FUNCTION_BLOCK PUBLIC FB_Step EXTENDS FB_Base
VAR_INPUT
END_VAR
VAR_OUTPUT
	nActStep	: UDINT := 0 ; // Active step
	bIdle		: BOOL	:= TRUE  ; // Stepper is idle (Step 0)
	bPaused		: BOOL 	:= FALSE ; // Stepper is paused
	bHold		: BOOL 	:= FALSE ; // Stepper is blocked for changes
	bSkipPause	: BOOL	:= FALSE ; // Pause function is skipped in this step 
	bResetting	: BOOL  := False ; // Reset is active
END_VAR
VAR
	nPreviousStep 	: UDINT ; // Previous active step
	nNextStep		: UDINT ; // Next step to activate
	nResetStep		: UDINT ; // step to which the stepper will go after reset
END_VAR

SetActiveStep();

METHOD PUBLIC CmdHold : BOOL
VAR_INPUT
END_VAR
bHold := TRUE ;

CmdHold := bHold;
END_METHOD

METHOD PUBLIC CmdNext : BOOL
VAR_INPUT
END_VAR
IF NOT bHold THEN 
	nNextStep := nActStep +	1 ;	
END_IF

CmdNext := TRUE ;
END_METHOD

METHOD PUBLIC CmdPrevious : BOOL
VAR_INPUT
END_VAR
IF NOT bHold THEN 
	nNextStep := nPreviousStep ;	
END_IF

CmdPrevious := TRUE ;
END_METHOD

METHOD PUBLIC CmdReset : BOOL
VAR_INPUT
END_VAR
bErrorActive := FALSE ;

IF nActStep <> nResetStep THEN 
	IF NOT bResetting THEN
		bResetting := TRUE ;
	ELSE
		nPreviousStep 	:= nActStep ;
		nNextStep		:= nResetStep ;
		nActStep 		:= nResetStep ;
		bResetting 		:= FALSE;
	END_IF
ELSE
	CmdReset := TRUE ; 
END_IF
END_METHOD

METHOD PUBLIC CmdToStep : BOOL
VAR_INPUT
	nStep	: UDINT ;
END_VAR
IF NOT bHold THEN 
	nNextStep := nStep ;
END_IF

CmdToStep := nNextStep = nStep ;
END_METHOD

METHOD PUBLIC Init : BOOL
VAR_INPUT
	// Location data for messages  
	nId			: UDINT ; // Identification number of object
	nParentId	: UDINT ; // Id of higher level If aplicable (0 = no parent)
	nResetStep	: UDINT ; // step to which the stepper wil go at reset
END_VAR
// ====== Calculate device id =====
	ExecIdentifyDevice(nId,nParentId,E_ComponentTypes.StepProgram);
	
// ===== set reset step ======
	nActStep 			:= nResetStep ;
	THIS^.nResetStep	:= nResetStep ;
END_METHOD

METHOD PRIVATE SetActiveStep : BOOL
VAR_INPUT
END_VAR
IF bResetting THEN 
	nPreviousStep 	:= nActStep ;
	nNextStep		:= nResetStep ;
	nActStep 		:= nResetStep ;
	bResetting 		:= FALSE; 
ELSIF bHold THEN 
	bHold 			:= FALSE ;
	RETURN; 
ELSIF bErrorActive THEN 
	stFault.Active			:= TRUE ;
	stFault.ComponentType	:= E_ComponentTypes.StepProgram ;
	stFault.Discription		:= CONCAT(sName, ' Invalid step state');
	stFault.FaultType		:= E_FaultTypes.FF;
	stFault.MessageNumber	:= E_MessageNumbers.FF_ComunicationFault;
ELSIF NOT bCmdPause OR bSkipPause THEN 
	IF nActStep <> nNextStep THEN 
		nPreviousStep 	:=	nActStep;	
		nActStep		:= 	nNextStep;
	END_IF
END_IF

bPaused 	:= bCmdPause ;	
bSkipPause 	:= FALSE ; 
bIdle 		:= nActStep = 0 ;
END_METHOD

METHOD Public SkipPause : BOOL
VAR_INPUT
END_VAR
bSkipPause := TRUE ;

SkipPause := true ;
END_METHOD

METHOD PUBLIC StepError : BOOL
VAR_INPUT
END_VAR
bErrorActive := TRUE ;
END_METHOD

END_FUNCTION_BLOCK

(* stored: Version 1.1.0.1, ProductVersion 3.1.4024.9
   POU FB_Step: Id {69b694f5-baa1-4f86-8caa-4a01db9ce8f8}, SpecialFunc None
   Folder Commands: Id {79421837-b695-48ee-b4a9-422180fd25e0}
   Method CmdHold: Id {8f8fda5c-2e20-4c09-b790-f4e6b77f96ee}
   Method CmdNext: Id {bc8d4796-dcaf-4c5e-bae9-87ceeef8aa99}
   Method CmdPrevious: Id {c2b04311-04d7-4f84-889d-0728cdacbfa0}
   Method CmdReset: Id {5aeae7cb-a474-4607-a12c-75090f5444bb}
   Method CmdToStep: Id {b9476a6f-d207-4362-99c9-73295ef1c21e}
   Method Init: Id {decf4df9-b1c5-4f84-8d5c-781cd3a12a56}
   Method SetActiveStep: Id {ff41807d-3ee0-4176-8aab-e544184b5717}
   Method SkipPause: Id {c383ca2b-0f6c-427f-82a9-3b5af80fb5b4}
   Method StepError: Id {65f1fa82-acef-4e31-8eee-11f570096477} *)
